Omron CX-Programmer project NewProject (CX-Programmer 9.51)

# PLC couter_demo: CP1L L

## Global symbols (name address type ; comment)
0.00 BOOL  ; UP
0.01 BOOL  ; DOWN
0.02 BOOL  ; RESET
0.03 BOOL  ; UP
0.04 BOOL  ; DOWN

## Program NewProgram1 (cyclic task 0)
Local symbols
P_off BOOL

### Section Section1

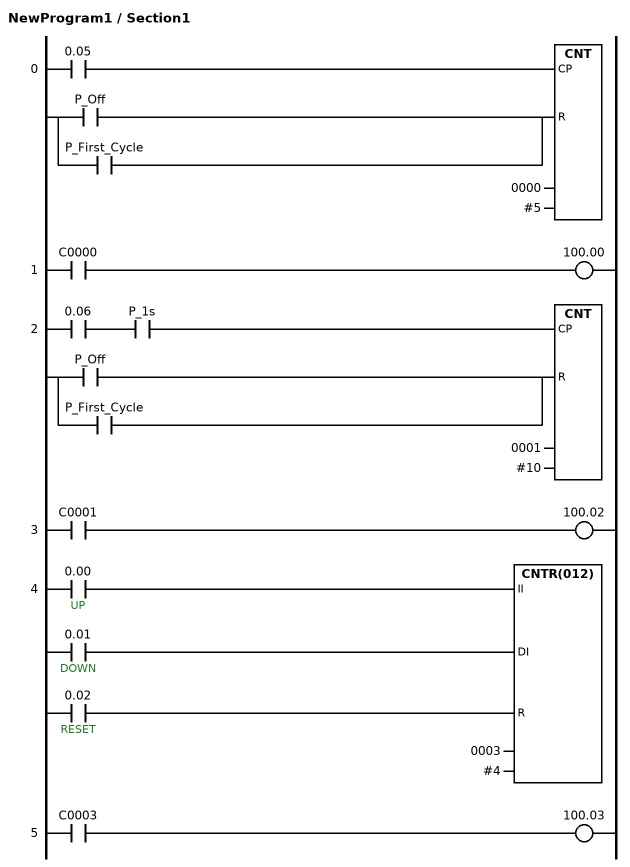
; rung 0
LD 0.05
LD P_Off
OR P_First_Cycle
CNT 0000 #5
; rung 1
LD C0000
OUT 100.00
; rung 2
LD 0.06
AND P_1s
LD P_Off
OR P_First_Cycle
CNT 0001 #10
; rung 3
LD C0001
OUT 100.02
; rung 4
LD 0.00  ; UP
LD 0.01  ; DOWN
LD 0.02  ; RESET
CNTR(012) 0003 #4
; rung 5
LD C0003
OUT 100.03

### Section END
; rung 0
END(001)